(* Schneider Machine Expert - Basic project Scada_tram_2, file version 2.7.0.0 *)
(* CompanyInformations: Name=tnd.jsc, PhoneNumber=+84988935902, Street=giai phong, City=ha noi, ZipCode=100000, State=58/88 giap nhi, Country=Viet Nam *)
(* ProjectInformations: Name=scada_tram 1&2 *)
(* UserInformations: LastName=lemanh, FirstName=tuan, PhoneNumber=+84988935902, CellNumber=+84988935902, Email=dientutnd@gmail.com, Street=giai phong, City=ha noi, ZipCode=100000, State=58/88 giap nhi, Country=Viet Nam *)

HARDWARE
  Cpu 0: TM221CE40R
  ModuleExtensionObject 0: TM3AQ4/G
  ModuleExtensionObject 1: TM3AI4/G
  EthernetConfiguration: NetworkName=M221, IpAllocationMode=FixedAddress, IpAddress=192.168.50.14, SubnetMask=255.255.255.0
  SerialLineConfiguration: Baud=Baud19200, Parity=ParityEven, DataBits=DataBits8, StopBits=StopBits1, PhysicalMedium=PhysicalMediumRs485, TransmissionMode=TransmissionModeModbusRtu, SlaveId=1, Addressing=SlaveAddressing
  MastTask: UsePeriodScanMode=false, PeriodScan=100
  FastTask: Period=255
  CpuBehavior: StartingMode=StartAsPreviousState, AutoSaveRamOnEeprom=true, WatchdogPeriod=250

SYMBOLS  (address, symbol, comment, settings)
  %M0       PROTECTED_PHASE
  %M1       LOW_CLEAN_WATER_POOL1
  %M2       LOW_CLEAN_WATER_POOL2
  %M3       LOW_WATER_POOL_INOX_1
  %M4       LOW_WATER_POOL_INOX_2
  %M5       POWER_EVETER_1
  %M6       POWER_EVETER_2
  %M7       RUN_EVETER_1
  %M8       RUN_EVETER_2
  %M9       RUN_PHÈN_3
  %M10      RUN_PHÈN_4
  %M11      RUN_KHUẤY_5
  %M12      RUN_KHUẤY_6
  %M13      NOT_USE
  %M14      ERROR_BT1
  %M15      ERROR_BT2
  %M16      ERROR_PHÈN_3
  %M17      ERROR_PHÈN_4
  %M18      ERROR_KHUẤY_5
  %M19      ERROR_KHUẤY_6
  %M21      RUN_COIL_PUMB1_REMOTE
  %M22      POWER_EL_1_REMOTE
  %M23      RUN_COIL_PUMB2_REMTOE
  %M24      POWER_EL_2_REMOTE
  %M31      RUN_COIL_PUMB1_AUTO
  %M32      POWER_EL_1_AUTO
  %M33      RUN_COIL_PUMB2_AUTO
  %M34      POWER_EL_2_AUTO
  %M41      J3
  %M42      J4
  %M43      K5
  %M44      K6
  %M51      PROTECT_P1
  %M52      PROTECT_P2
  %M53      CHE_DO_AUTO
  %S6       SB_TB1S  "Time base of 1 s generated by an internal clock"
  %MW1      AO_PUMB_1
  %MW2      AO_PUMB_2
  %MW3      SET_PERSURE
  %MW4      AI_PIPE
  %MW10     LOGIC_PUMB_1
  %MW13     MAP_SET_PERSURE
  %TM0      TIMER_RUN_PUMB11  "Time delay"  [Preset=10, Base=OneSecond]
  %TM1      TIMER_OFF_EVETER1  [Type=TOF, Preset=40, Base=OneSecond]
  %TM2      TIMER_RUN_PUMB2  [Preset=10, Base=OneSecond]
  %TM3      TIMER_OFF_EVETER2  [Type=TOF, Preset=40, Base=OneSecond]
  %TM4      TIMER_RESET_PUMB_2_AUTO  [Type=TOF, Preset=20, Base=OneSecond]
  %Q0.0     SP1
  %Q0.1     PE1
  %Q0.2     SP2
  %Q0.3     PE2
  %Q0.4     RUN_JAVEN_3
  %Q0.5     RUN_JAVEN_4
  %Q0.6     SK5
  %Q0.7     SK6
  %QW1.1    ANALOG_OUTPUT_EL1  [Type=Type_4_20mA, Scope=Scope_Customized, Minimum=4000, Maximum=20000]
  %QW1.2    ANALOG_OUTPUT_EL2  [Type=Type_4_20mA, Scope=Scope_Customized, Minimum=4000, Maximum=20000]
  %IW2.0    PERSURE_PIPE  [Type=Type_4_20mA, Scope=Scope_Customized, Minimum=4000, Maximum=20000]

POU Add DI to SingleCoil
  (* SectionNumber=1 *)

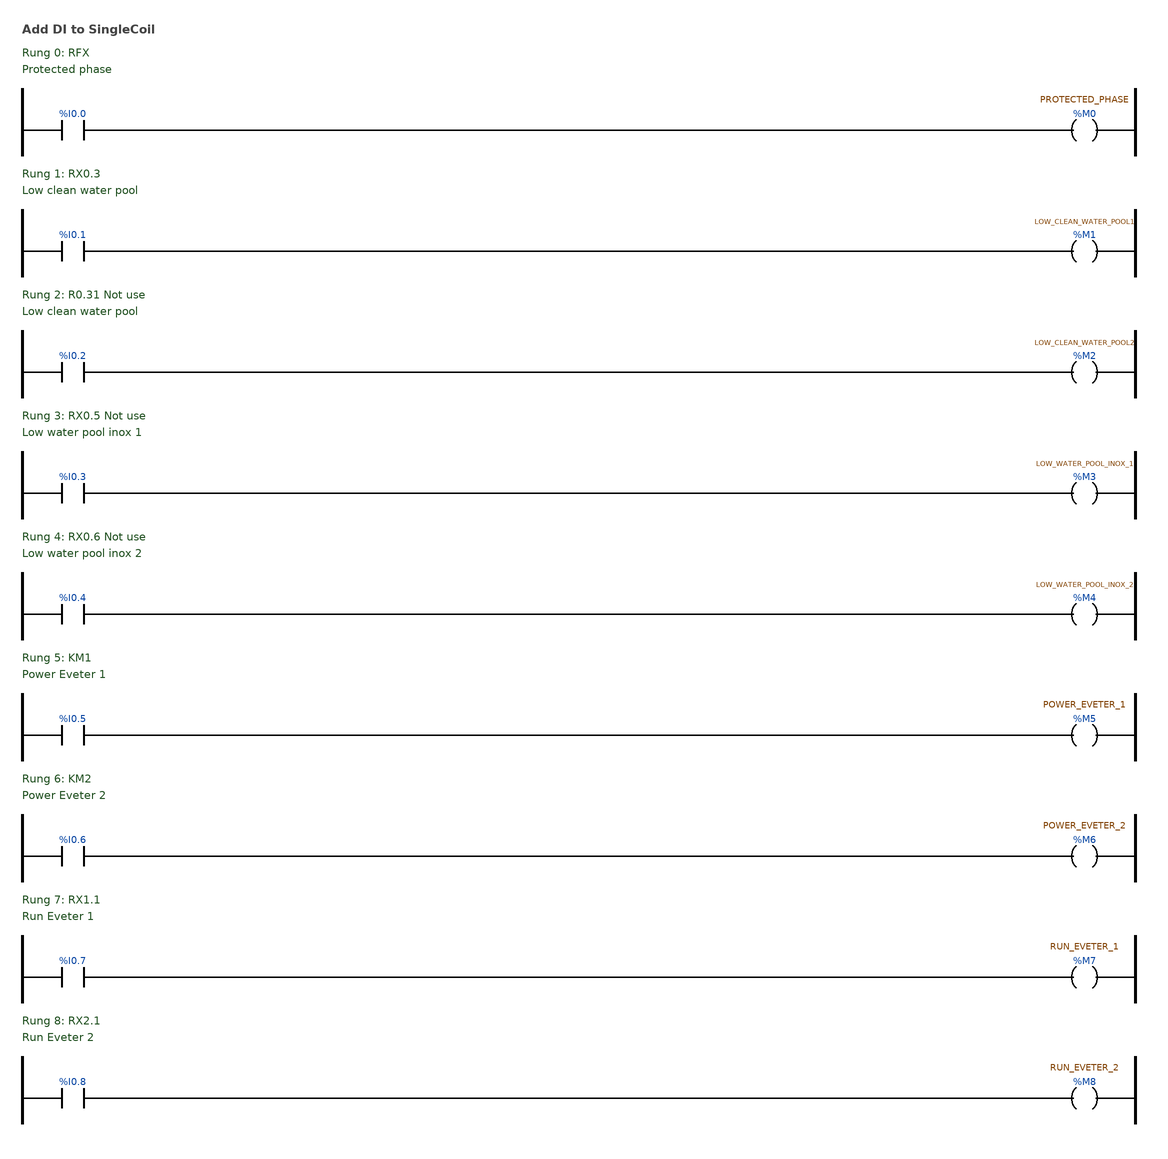

// Rung 0: RFX
// Protected phase
  LD %I0.0
  ST %M0                  (* PROTECTED_PHASE *)
  // as ST:
  //   PROTECTED_PHASE := %I0.0;

// Rung 1: RX0.3
// Low clean water pool
  LD %I0.1
  ST %M1                  (* LOW_CLEAN_WATER_POOL1 *)
  // as ST:
  //   LOW_CLEAN_WATER_POOL1 := %I0.1;

// Rung 2: R0.31 Not use
// Low clean water pool
  LD %I0.2
  ST %M2                  (* LOW_CLEAN_WATER_POOL2 *)
  // as ST:
  //   LOW_CLEAN_WATER_POOL2 := %I0.2;

// Rung 3: RX0.5 Not use
// Low water pool inox 1
  LD %I0.3
  ST %M3                  (* LOW_WATER_POOL_INOX_1 *)
  // as ST:
  //   LOW_WATER_POOL_INOX_1 := %I0.3;

// Rung 4: RX0.6 Not use
// Low water pool inox 2
  LD %I0.4
  ST %M4                  (* LOW_WATER_POOL_INOX_2 *)
  // as ST:
  //   LOW_WATER_POOL_INOX_2 := %I0.4;

// Rung 5: KM1
// Power Eveter 1
  LD %I0.5
  ST %M5                  (* POWER_EVETER_1 *)
  // as ST:
  //   POWER_EVETER_1 := %I0.5;

// Rung 6: KM2
// Power Eveter 2
  LD %I0.6
  ST %M6                  (* POWER_EVETER_2 *)
  // as ST:
  //   POWER_EVETER_2 := %I0.6;

// Rung 7: RX1.1
// Run Eveter 1
  LD %I0.7
  ST %M7                  (* RUN_EVETER_1 *)
  // as ST:
  //   RUN_EVETER_1 := %I0.7;

// Rung 8: RX2.1
// Run Eveter 2
  LD %I0.8
  ST %M8                  (* RUN_EVETER_2 *)
  // as ST:
  //   RUN_EVETER_2 := %I0.8;

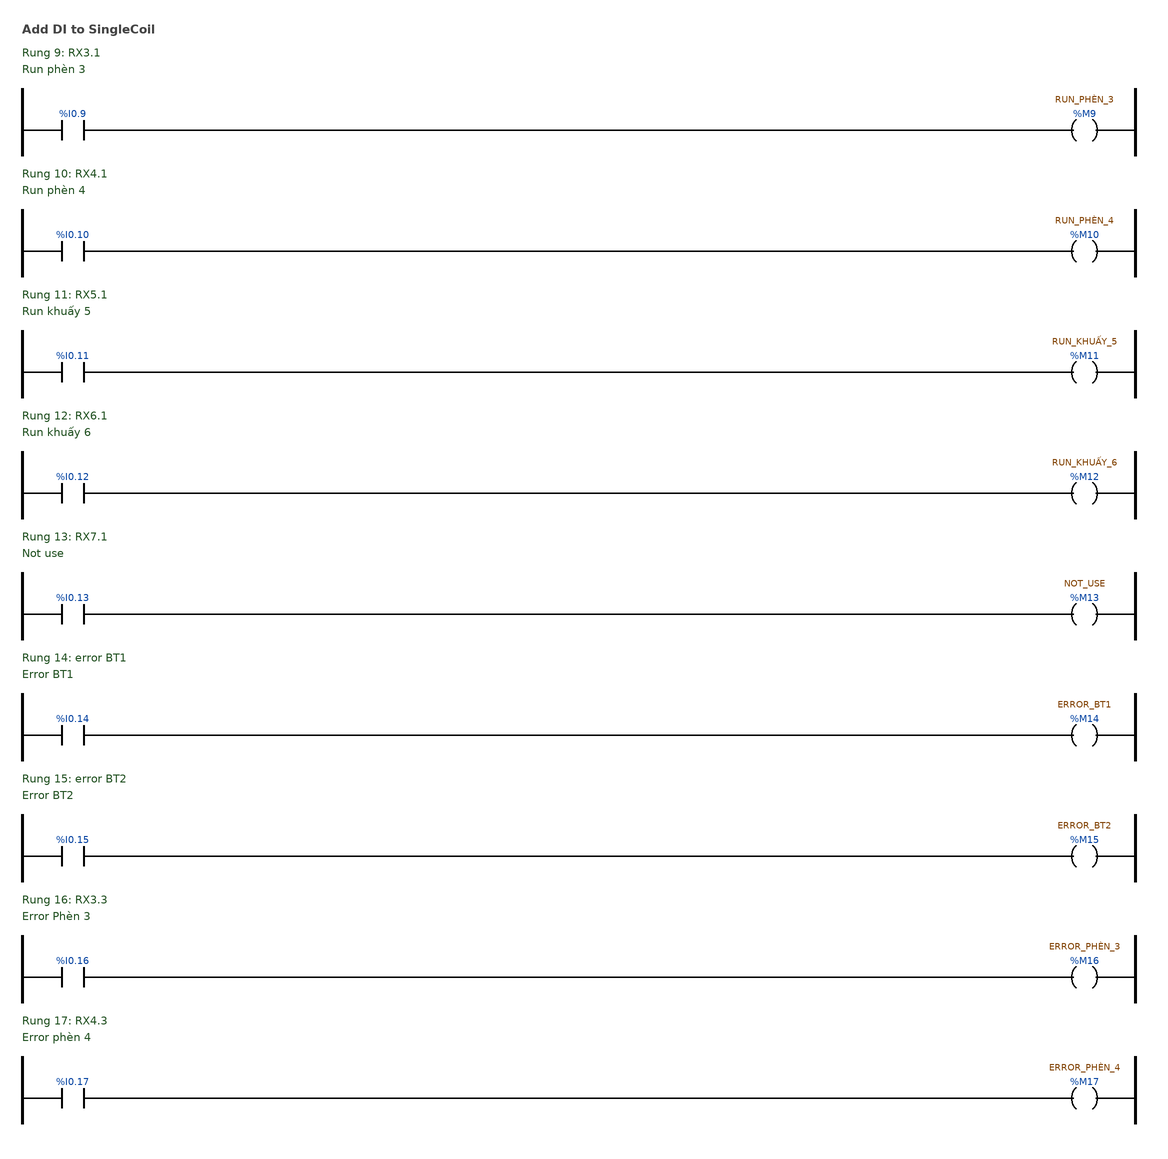

// Rung 9: RX3.1
// Run phèn 3
  LD %I0.9
  ST %M9                  (* RUN_PHÈN_3 *)
  // as ST:
  //   RUN_PHÈN_3 := %I0.9;

// Rung 10: RX4.1
// Run phèn 4
  LD %I0.10
  ST %M10                 (* RUN_PHÈN_4 *)
  // as ST:
  //   RUN_PHÈN_4 := %I0.10;

// Rung 11: RX5.1
// Run khuấy 5
  LD %I0.11
  ST %M11                 (* RUN_KHUẤY_5 *)
  // as ST:
  //   RUN_KHUẤY_5 := %I0.11;

// Rung 12: RX6.1
// Run khuấy 6
  LD %I0.12
  ST %M12                 (* RUN_KHUẤY_6 *)
  // as ST:
  //   RUN_KHUẤY_6 := %I0.12;

// Rung 13: RX7.1
// Not use
  LD %I0.13
  ST %M13                 (* NOT_USE *)
  // as ST:
  //   NOT_USE := %I0.13;

// Rung 14: error BT1
// Error BT1
  LD %I0.14
  ST %M14                 (* ERROR_BT1 *)
  // as ST:
  //   ERROR_BT1 := %I0.14;

// Rung 15: error BT2
// Error BT2
  LD %I0.15
  ST %M15                 (* ERROR_BT2 *)
  // as ST:
  //   ERROR_BT2 := %I0.15;

// Rung 16: RX3.3
// Error Phèn 3
  LD %I0.16
  ST %M16                 (* ERROR_PHÈN_3 *)
  // as ST:
  //   ERROR_PHÈN_3 := %I0.16;

// Rung 17: RX4.3
// Error phèn 4
  LD %I0.17
  ST %M17                 (* ERROR_PHÈN_4 *)
  // as ST:
  //   ERROR_PHÈN_4 := %I0.17;

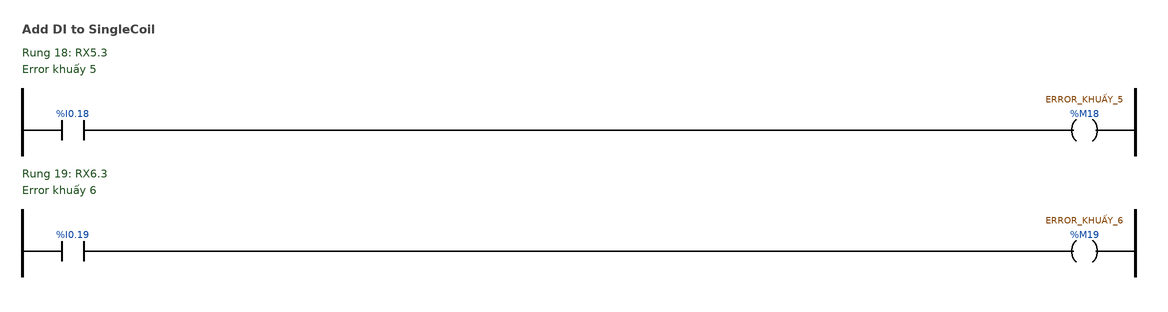

// Rung 18: RX5.3
// Error khuấy 5
  LD %I0.18
  ST %M18                 (* ERROR_KHUẤY_5 *)
  // as ST:
  //   ERROR_KHUẤY_5 := %I0.18;

// Rung 19: RX6.3
// Error khuấy 6
  LD %I0.19
  ST %M19                 (* ERROR_KHUẤY_6 *)
  // as ST:
  //   ERROR_KHUẤY_6 := %I0.19;

POU Remote Control Pump
  (* SectionNumber=2 *)

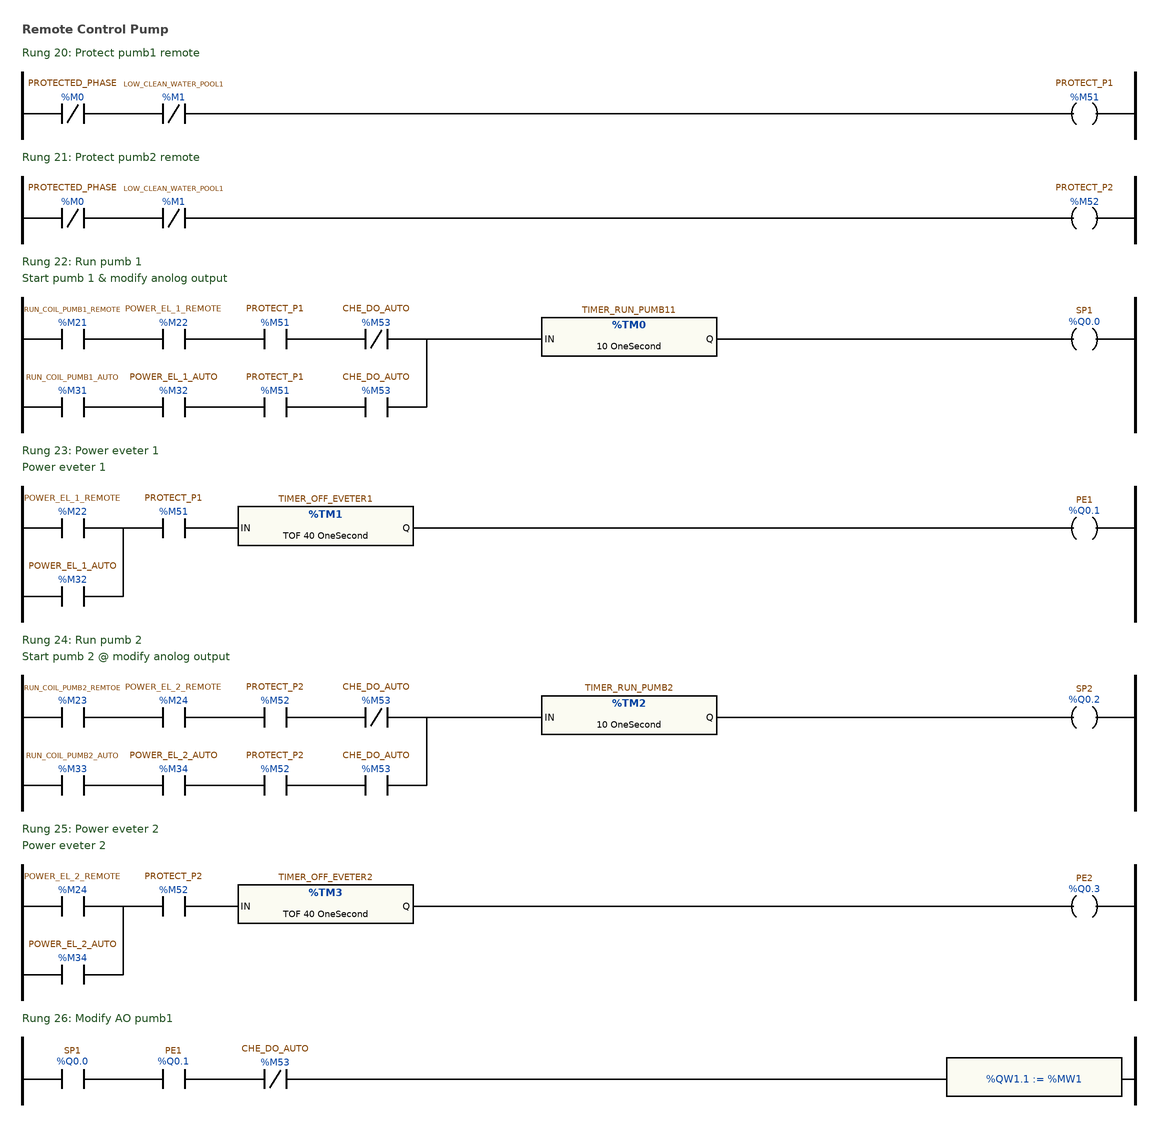

// Rung 20: Protect pumb1 remote
  LDN %M0                 (* PROTECTED_PHASE *)
  ANDN %M1                (* LOW_CLEAN_WATER_POOL1 *)
  ST %M51                 (* PROTECT_P1 *)
  // as ST:
  //   PROTECT_P1 := NOT PROTECTED_PHASE AND NOT LOW_CLEAN_WATER_POOL1;

// Rung 21: Protect pumb2 remote
  LDN %M0                 (* PROTECTED_PHASE *)
  ANDN %M1                (* LOW_CLEAN_WATER_POOL1 *)
  ST %M52                 (* PROTECT_P2 *)
  // as ST:
  //   PROTECT_P2 := NOT PROTECTED_PHASE AND NOT LOW_CLEAN_WATER_POOL1;

// Rung 22: Run pumb 1
// Start pumb 1 & modify anolog output
  BLK %TM0                (* TIMER_RUN_PUMB11 *)
  LD %M21                 (* RUN_COIL_PUMB1_REMOTE *)
  AND %M22                (* POWER_EL_1_REMOTE *)
  AND %M51                (* PROTECT_P1 *)
  ANDN %M53               (* CHE_DO_AUTO *)
  OR( %M31                (* RUN_COIL_PUMB1_AUTO *)
  AND %M32                (* POWER_EL_1_AUTO *)
  AND %M51                (* PROTECT_P1 *)
  AND %M53                (* CHE_DO_AUTO *)
  )
  IN
  OUT_BLK
  LD Q
  ST %Q0.0                (* SP1 *)
  END_BLK
  // as ST:
  //   TIMER_RUN_PUMB11(IN := RUN_COIL_PUMB1_REMOTE AND POWER_EL_1_REMOTE AND PROTECT_P1 AND NOT CHE_DO_AUTO OR RUN_COIL_PUMB1_AUTO AND POWER_EL_1_AUTO AND PROTECT_P1 AND CHE_DO_AUTO);
  //   SP1 := TIMER_RUN_PUMB11.Q;

// Rung 23: Power eveter 1
// Power eveter 1
  BLK %TM1                (* TIMER_OFF_EVETER1 *)
  LD %M22                 (* POWER_EL_1_REMOTE *)
  OR %M32                 (* POWER_EL_1_AUTO *)
  AND %M51                (* PROTECT_P1 *)
  IN
  OUT_BLK
  LD Q
  ST %Q0.1                (* PE1 *)
  END_BLK
  // as ST:
  //   TIMER_OFF_EVETER1(IN := (POWER_EL_1_REMOTE OR POWER_EL_1_AUTO) AND PROTECT_P1);
  //   PE1 := TIMER_OFF_EVETER1.Q;

// Rung 24: Run pumb 2
// Start pumb 2 @ modify anolog output
  BLK %TM2                (* TIMER_RUN_PUMB2 *)
  LD %M23                 (* RUN_COIL_PUMB2_REMTOE *)
  AND %M24                (* POWER_EL_2_REMOTE *)
  AND %M52                (* PROTECT_P2 *)
  ANDN %M53               (* CHE_DO_AUTO *)
  OR( %M33                (* RUN_COIL_PUMB2_AUTO *)
  AND %M34                (* POWER_EL_2_AUTO *)
  AND %M52                (* PROTECT_P2 *)
  AND %M53                (* CHE_DO_AUTO *)
  )
  IN
  OUT_BLK
  LD Q
  ST %Q0.2                (* SP2 *)
  END_BLK
  // as ST:
  //   TIMER_RUN_PUMB2(IN := RUN_COIL_PUMB2_REMTOE AND POWER_EL_2_REMOTE AND PROTECT_P2 AND NOT CHE_DO_AUTO OR RUN_COIL_PUMB2_AUTO AND POWER_EL_2_AUTO AND PROTECT_P2 AND CHE_DO_AUTO);
  //   SP2 := TIMER_RUN_PUMB2.Q;

// Rung 25: Power eveter 2
// Power eveter 2
  BLK %TM3                (* TIMER_OFF_EVETER2 *)
  LD %M24                 (* POWER_EL_2_REMOTE *)
  OR %M34                 (* POWER_EL_2_AUTO *)
  AND %M52                (* PROTECT_P2 *)
  IN
  OUT_BLK
  LD Q
  ST %Q0.3                (* PE2 *)
  END_BLK
  // as ST:
  //   TIMER_OFF_EVETER2(IN := (POWER_EL_2_REMOTE OR POWER_EL_2_AUTO) AND PROTECT_P2);
  //   PE2 := TIMER_OFF_EVETER2.Q;

// Rung 26: Modify AO pumb1
  LD %Q0.0                (* SP1 *)
  AND %Q0.1               (* PE1 *)
  ANDN %M53               (* CHE_DO_AUTO *)
  [ %QW1.1 := %MW1 ]      (* ANALOG_OUTPUT_EL1, AO_PUMB_1 *)
  // as ST:
  //   IF SP1 AND PE1 AND NOT CHE_DO_AUTO THEN ANALOG_OUTPUT_EL1 := AO_PUMB_1; END_IF;

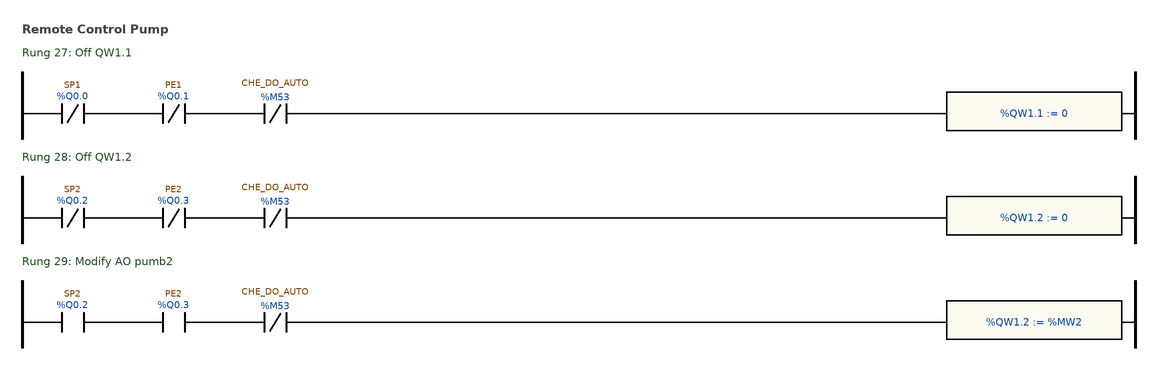

// Rung 27: Off QW1.1
  LDN %Q0.0               (* SP1 *)
  ANDN %Q0.1              (* PE1 *)
  ANDN %M53               (* CHE_DO_AUTO *)
  [ %QW1.1 := 0 ]         (* ANALOG_OUTPUT_EL1 *)
  // as ST:
  //   IF NOT SP1 AND NOT PE1 AND NOT CHE_DO_AUTO THEN ANALOG_OUTPUT_EL1 := 0; END_IF;

// Rung 28: Off QW1.2
  LDN %Q0.2               (* SP2 *)
  ANDN %Q0.3              (* PE2 *)
  ANDN %M53               (* CHE_DO_AUTO *)
  [ %QW1.2 := 0 ]         (* ANALOG_OUTPUT_EL2 *)
  // as ST:
  //   IF NOT SP2 AND NOT PE2 AND NOT CHE_DO_AUTO THEN ANALOG_OUTPUT_EL2 := 0; END_IF;

// Rung 29: Modify AO pumb2
  LD %Q0.2                (* SP2 *)
  AND %Q0.3               (* PE2 *)
  ANDN %M53               (* CHE_DO_AUTO *)
  [ %QW1.2 := %MW2 ]      (* ANALOG_OUTPUT_EL2, AO_PUMB_2 *)
  // as ST:
  //   IF SP2 AND PE2 AND NOT CHE_DO_AUTO THEN ANALOG_OUTPUT_EL2 := AO_PUMB_2; END_IF;

POU Auto Control Pumb
  (* SectionNumber=3 *)

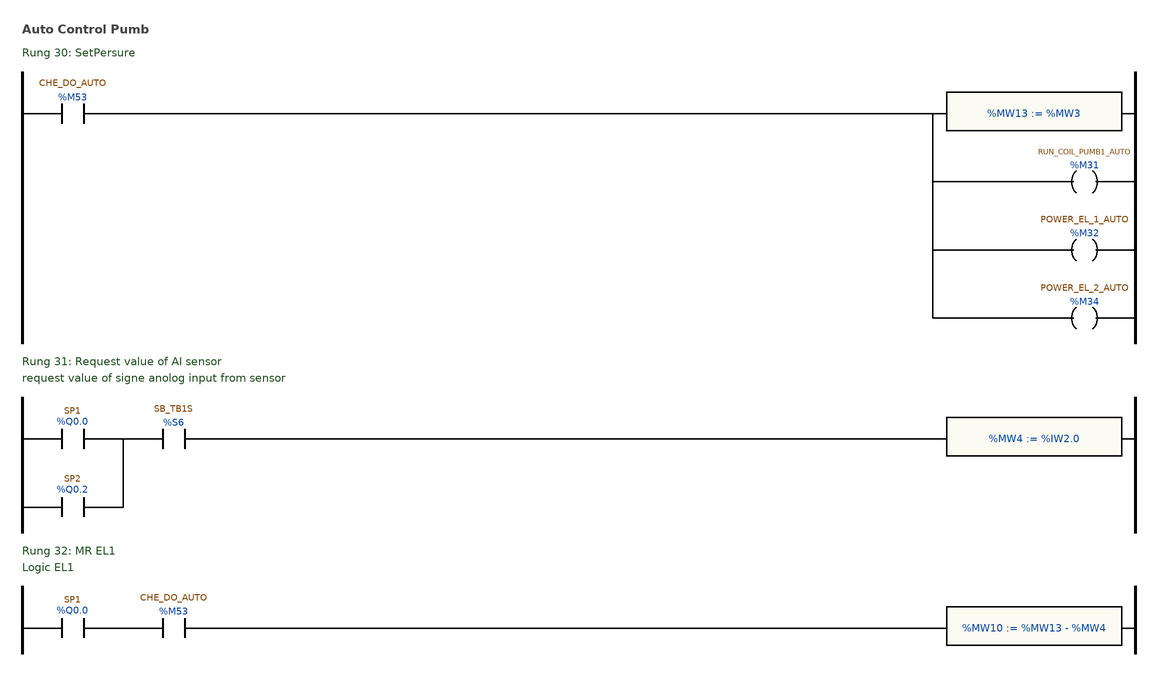

// Rung 30: SetPersure
  LD %M53                 (* CHE_DO_AUTO *)
  [ %MW13 := %MW3 ]       (* MAP_SET_PERSURE, SET_PERSURE *)
  ST %M31                 (* RUN_COIL_PUMB1_AUTO *)
  ST %M32                 (* POWER_EL_1_AUTO *)
  ST %M34                 (* POWER_EL_2_AUTO *)
  // as ST:
  //   IF CHE_DO_AUTO THEN MAP_SET_PERSURE := SET_PERSURE; END_IF;
  //   RUN_COIL_PUMB1_AUTO := CHE_DO_AUTO;
  //   POWER_EL_1_AUTO := CHE_DO_AUTO;
  //   POWER_EL_2_AUTO := CHE_DO_AUTO;

// Rung 31: Request value of AI sensor
// request value of signe anolog input from sensor
  LD %Q0.0                (* SP1 *)
  OR %Q0.2                (* SP2 *)
  AND %S6                 (* SB_TB1S *)
  [ %MW4 := %IW2.0 ]      (* AI_PIPE, PERSURE_PIPE *)
  // as ST:
  //   IF (SP1 OR SP2) AND SB_TB1S THEN AI_PIPE := PERSURE_PIPE; END_IF;

// Rung 32: MR EL1
// Logic EL1
  LD %Q0.0                (* SP1 *)
  AND %M53                (* CHE_DO_AUTO *)
  [ %MW10 := %MW13 - %MW4 ](* LOGIC_PUMB_1, MAP_SET_PERSURE, AI_PIPE *)
  // as ST:
  //   IF SP1 AND CHE_DO_AUTO THEN LOGIC_PUMB_1 := MAP_SET_PERSURE - AI_PIPE; END_IF;

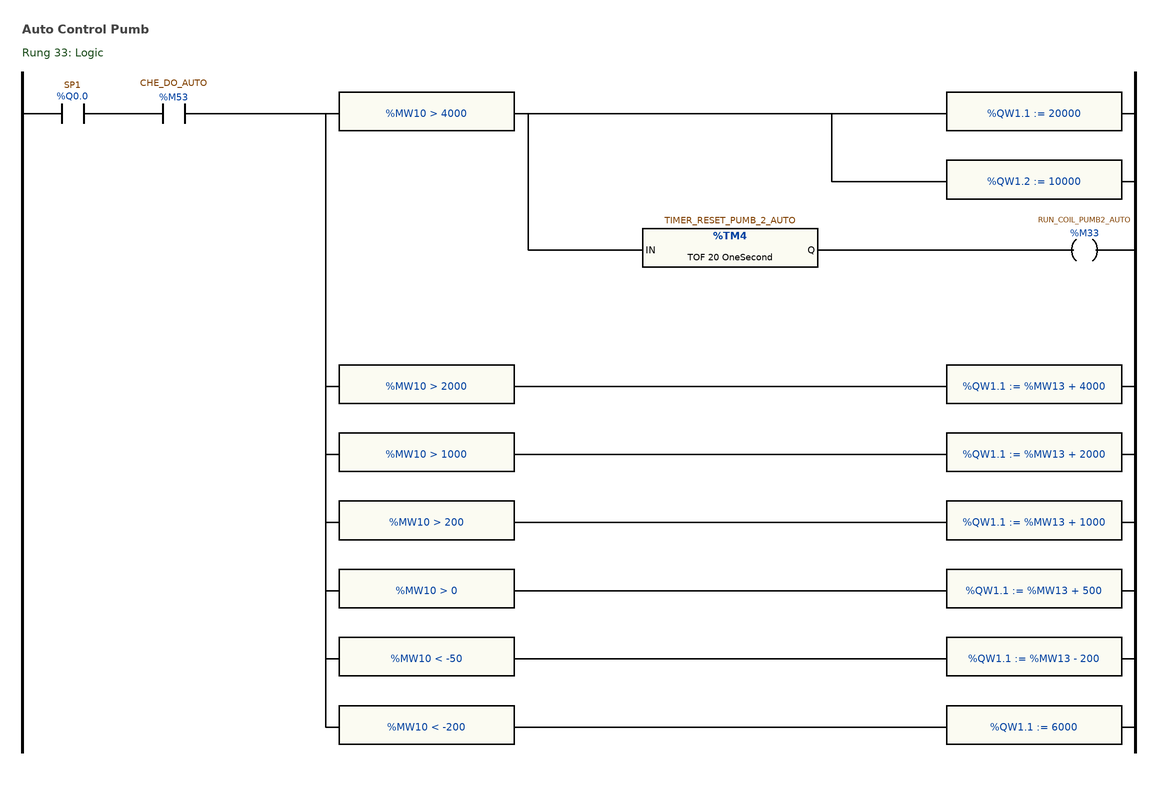

// Rung 33: Logic
  LD 1
  MULTIFB
  LD 1
  AND %Q0.0               (* SP1 *)
  AND %M53                (* CHE_DO_AUTO *)
  ST %MW2009:X0
  LD %MW2009:X0
  AND [ %MW10 > 4000 ]    (* LOGIC_PUMB_1 *)
  ST %MW2009:X1
  LD %MW2009:X1
  [ %QW1.1 := 20000 ]     (* ANALOG_OUTPUT_EL1 *)
  [ %QW1.2 := 10000 ]     (* ANALOG_OUTPUT_EL2 *)
  BLK %TM4                (* TIMER_RESET_PUMB_2_AUTO *)
  LD %MW2009:X1
  IN
  OUT_BLK
  LD Q
  ST %M33                 (* RUN_COIL_PUMB2_AUTO *)
  END_BLK
  LD %MW2009:X0
  MPS
  AND [ %MW10 > 2000 ]    (* LOGIC_PUMB_1 *)
  [ %QW1.1 := %MW13 + 4000 ](* ANALOG_OUTPUT_EL1, MAP_SET_PERSURE *)
  MRD
  AND [ %MW10 > 1000 ]    (* LOGIC_PUMB_1 *)
  [ %QW1.1 := %MW13 + 2000 ](* ANALOG_OUTPUT_EL1, MAP_SET_PERSURE *)
  MRD
  AND [ %MW10 > 200 ]     (* LOGIC_PUMB_1 *)
  [ %QW1.1 := %MW13 + 1000 ](* ANALOG_OUTPUT_EL1, MAP_SET_PERSURE *)
  MRD
  AND [ %MW10 > 0 ]       (* LOGIC_PUMB_1 *)
  [ %QW1.1 := %MW13 + 500 ](* ANALOG_OUTPUT_EL1, MAP_SET_PERSURE *)
  MRD
  AND [ %MW10 < -50 ]     (* LOGIC_PUMB_1 *)
  [ %QW1.1 := %MW13 - 200 ](* ANALOG_OUTPUT_EL1, MAP_SET_PERSURE *)
  MPP
  AND [ %MW10 < -200 ]    (* LOGIC_PUMB_1 *)
  [ %QW1.1 := 6000 ]      (* ANALOG_OUTPUT_EL1 *)
  MULTIFB
  // as ST:
  //   IF SP1 AND CHE_DO_AUTO AND LOGIC_PUMB_1 > 4000 THEN ANALOG_OUTPUT_EL1 := 20000; END_IF;
  //   IF SP1 AND CHE_DO_AUTO AND LOGIC_PUMB_1 > 4000 THEN ANALOG_OUTPUT_EL2 := 10000; END_IF;
  //   TIMER_RESET_PUMB_2_AUTO(IN := SP1 AND CHE_DO_AUTO AND LOGIC_PUMB_1 > 4000);
  //   RUN_COIL_PUMB2_AUTO := TIMER_RESET_PUMB_2_AUTO.Q;
  //   IF SP1 AND CHE_DO_AUTO AND LOGIC_PUMB_1 > 2000 THEN ANALOG_OUTPUT_EL1 := MAP_SET_PERSURE + 4000; END_IF;
  //   IF SP1 AND CHE_DO_AUTO AND LOGIC_PUMB_1 > 1000 THEN ANALOG_OUTPUT_EL1 := MAP_SET_PERSURE + 2000; END_IF;
  //   IF SP1 AND CHE_DO_AUTO AND LOGIC_PUMB_1 > 200 THEN ANALOG_OUTPUT_EL1 := MAP_SET_PERSURE + 1000; END_IF;
  //   IF SP1 AND CHE_DO_AUTO AND LOGIC_PUMB_1 > 0 THEN ANALOG_OUTPUT_EL1 := MAP_SET_PERSURE + 500; END_IF;
  //   IF SP1 AND CHE_DO_AUTO AND LOGIC_PUMB_1 < -50 THEN ANALOG_OUTPUT_EL1 := MAP_SET_PERSURE - 200; END_IF;
  //   IF SP1 AND CHE_DO_AUTO AND LOGIC_PUMB_1 < -200 THEN ANALOG_OUTPUT_EL1 := 6000; END_IF;

POU ControPumb3-6
  (* SectionNumber=4 *)

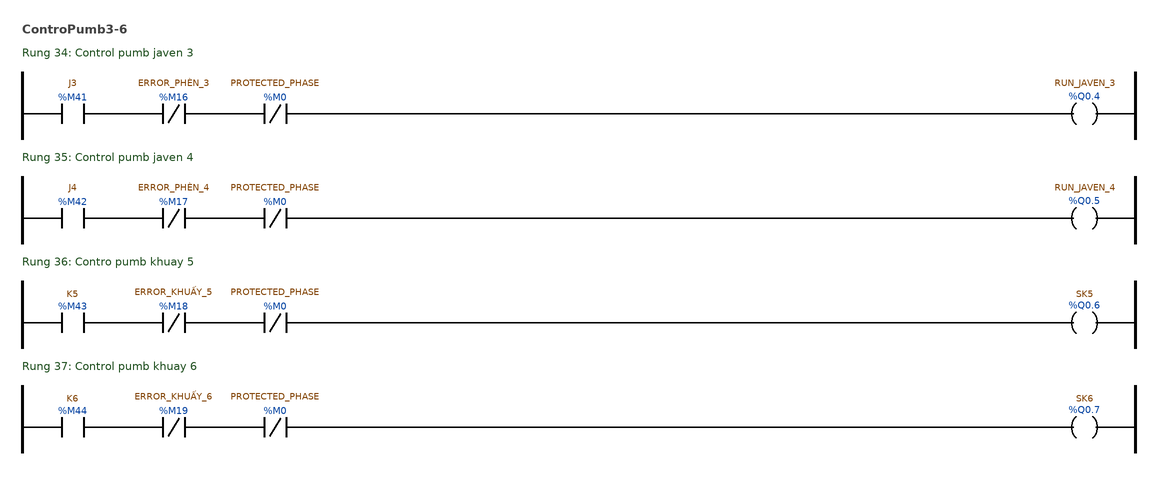

// Rung 34: Control pumb javen 3
  LD %M41                 (* J3 *)
  ANDN %M16               (* ERROR_PHÈN_3 *)
  ANDN %M0                (* PROTECTED_PHASE *)
  ST %Q0.4                (* RUN_JAVEN_3 *)
  // as ST:
  //   RUN_JAVEN_3 := J3 AND NOT ERROR_PHÈN_3 AND NOT PROTECTED_PHASE;

// Rung 35: Control pumb javen 4
  LD %M42                 (* J4 *)
  ANDN %M17               (* ERROR_PHÈN_4 *)
  ANDN %M0                (* PROTECTED_PHASE *)
  ST %Q0.5                (* RUN_JAVEN_4 *)
  // as ST:
  //   RUN_JAVEN_4 := J4 AND NOT ERROR_PHÈN_4 AND NOT PROTECTED_PHASE;

// Rung 36: Contro pumb khuay 5
  LD %M43                 (* K5 *)
  ANDN %M18               (* ERROR_KHUẤY_5 *)
  ANDN %M0                (* PROTECTED_PHASE *)
  ST %Q0.6                (* SK5 *)
  // as ST:
  //   SK5 := K5 AND NOT ERROR_KHUẤY_5 AND NOT PROTECTED_PHASE;

// Rung 37: Control pumb khuay 6
  LD %M44                 (* K6 *)
  ANDN %M19               (* ERROR_KHUẤY_6 *)
  ANDN %M0                (* PROTECTED_PHASE *)
  ST %Q0.7                (* SK6 *)
  // as ST:
  //   SK6 := K6 AND NOT ERROR_KHUẤY_6 AND NOT PROTECTED_PHASE;
